// TIA Portal V16 export
// export: Created 2020-03-21T17:35:44.067612Z, ExportSetting None, DisplayName Totally Integrated Automation Portal, DisplayVersion V16, DisplayName TIA Portal Version Control Interface, DisplayVersion V16, DisplayName TIA Portal Openness, DisplayVersion V16, DisplayName SINAMICS Startdrive Advanced, DisplayVersion V16, DisplayName SINAMICS Startdrive G130, G150, S120, S150, SINAMICS MV, S210, DisplayVersion V16, DisplayName SINAMICS Startdrive G110M, G120, G120C, G120D, G120P, DisplayVersion V16, DisplayName STEP 7 Professional, DisplayVersion V16, DisplayName STEP 7 Safety, DisplayVersion V16, DisplayName WinCC Advanced, DisplayVersion V16
FUNCTION "Block_1" : Void   // FC1, LAD
TITLE = Block Title
{ S7_Optimized_Access := 'TRUE' }
// Block Kommentar 1
// stored: SetENOAutomatically false
BEGIN

REGION Network 1: Netzwerk 1
   // Netzwerk Kommentar 1
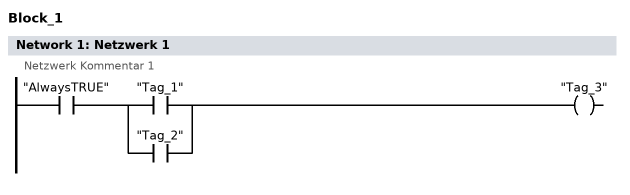
   RUNG wire#powerrail
      Contact( "AlwaysTRUE" )
      wire#w1
      Contact( "Tag_1" )
      wire#w2
      Coil( "Tag_3" )
   END_RUNG
   RUNG wire#w1
      Contact( "Tag_2" )
   END_RUNG wire#w2
   // the same network as SCL:
   "Tag_3" := "AlwaysTRUE" AND ("Tag_1" OR "Tag_2");
END_REGION
END_FUNCTION
